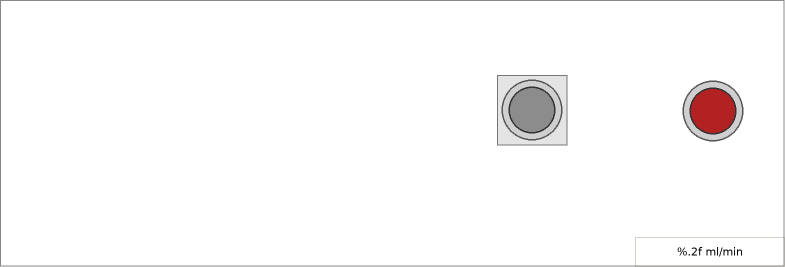
VISUALIZATION Visualization  // 785x267
    Lamp1 (678,76 70x70), variable: MAIN.FuelMeasurement1.timerRunning, style: Lamp-Lamp1-Red
    Textfield (635,237 150x30), "%.2f ml/min", text variable: MAIN.FuelVolumePerSec
    PushSwitch (497,75 70x70), variable: GVL.bStartMeasurement, behaviour: TAP, style: Switch-PushSwitch-Gray
END_VISUALIZATION

(* stored: Version 1.1.0.1, ProductVersion 3.1.4024.13
   Visu Visualization: Id {f1541733-5b18-4a5e-8843-4af1c3c30d78} *)
